FUNCTION_BLOCK SS3_Camera (* Basic FB with empty ECC *)
  (* Standard: 61499-2 *)
  (* Version 1.0, 2025-08-24, DEVIASH *)
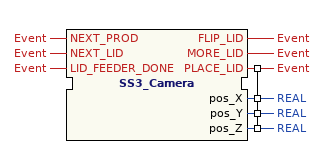
  EVENT_INPUT
    NEXT_PROD;
    NEXT_LID;
    LID_FEEDER_DONE;
  END_EVENT
  EVENT_OUTPUT
    FLIP_LID;
    MORE_LID;
    PLACE_LID WITH pos_X, pos_Y, pos_Z;
  END_EVENT
  VAR_OUTPUT
    pos_X : REAL;
    pos_Y : REAL;
    pos_Z : REAL;
  END_VAR
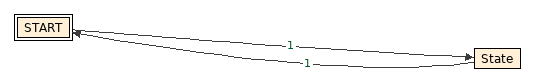
  EC_STATES
    START; (* Initial State *)
    State;
  END_STATES
  EC_TRANSITIONS
    START TO State := 1;
    State TO START := 1;
  END_TRANSITIONS
END_FUNCTION_BLOCK
